PROGRAM P_control_global
VAR
END_VAR

P_feedback_calculation();

IF GVL_P_CONTROL.P_loop_type THEN
	//Open loop control case
	GVL_P_CONTROL.P_block_output:= GVL_P_CONTROL.P_block_input;
ELSE
	//Closed loop control case
END_IF

END_PROGRAM

(* stored: Version 1.1.0.1, ProductVersion 3.1.4024.11
   POU P_control_global: Id {a7a9c095-8cda-4718-9941-39253879d8f5}, SpecialFunc None *)
